{attribute 'GeneratedUsingTerminal: EL2521-0124-0018'}
{attribute addProperty BoxType "EL2521-0124-0018"}
{attribute addProperty Description "EL2521-0124 1Ch. Pulse Train 24V DC Output Capture/Compare"}
{attribute addProperty Physics "KK"}
{attribute addProperty Id "PTO_StatusAT %I*PTO_Status_E0EB10E85ENC_Status_compactAT %I*ENC_Status_compact_3C6E2C4411PLS_StatusAT %I*PLS_Status_70E7A1E24PTO_ControlAT %Q*PTO_Control_9287F8E45PTO_Target_compactAT %Q*PTO_Target_compact_5C359F7D2ENC_Control_compactAT %Q*ENC_Control_compact_2E82BC435PLS_Control_compactAT %Q*PLS_Control_compact_CD6E44DE6WcStateAT %I*WcState_9091E0EB2InfoDataAT %I*InfoData_32EB74EA10"}
{attribute addProperty CRC "776196916"}
{attribute addProperty Size "50"}
TYPE EL2521_2E43D334 EXTENDS EtcSlaveTerminalBase_947E5A46 :
STRUCT
	{attribute addProperty Name "PTO_Status"}
	PTO_Status : PTO_Status_E0EB10E8;
	{attribute addProperty Name "ENC_Status_compact"}
	ENC_Status_compact : ENC_Status_compact_3C6E2C44;
	{attribute addProperty Name "PLS_Status"}
	PLS_Status : PLS_Status_70E7A1E2;
	{attribute addProperty Name "PTO_Control"}
	PTO_Control : PTO_Control_9287F8E4;
	{attribute addProperty Name "PTO_Target_compact"}
	PTO_Target_compact : PTO_Target_compact_5C359F7D;
	{attribute addProperty Name "ENC_Control_compact"}
	ENC_Control_compact : ENC_Control_compact_2E82BC43;
	{attribute addProperty Name "PLS_Control_compact"}
	PLS_Control_compact : PLS_Control_compact_CD6E44DE;
	{attribute addProperty Name "WcState"}
	WcState : WcState_9091E0EB;
	{attribute addProperty Name "InfoData"}
	InfoData : InfoData_32EB74EA;
END_STRUCT
END_TYPE

(* stored: Version 1.2.0.0, ProductVersion 3.1.4024.9
   DUT EL2521_2E43D334: Id {cf1d3700-59b4-4663-b5d0-cd147b47de77} *)
